// TIA Portal V17 export
// export: Created 2025-06-26T07:49:37.0369601Z, ExportSetting WithDefaults, DisplayName Totally Integrated Automation Portal, DisplayVersion V17 Update 8, DisplayName TIA Portal Openness, DisplayVersion V17 Update 8, DisplayName TIA Portal Version Control Interface, DisplayVersion V17, DisplayName STEP 7 Professional, DisplayVersion V17 Update 8, DisplayName STEP 7 Safety, DisplayVersion V17 Update 6, DisplayName WinCC Advanced, DisplayVersion V17 Update 8
FUNCTION "Control" : Void   // FC3, FBD
TITLE = Sequencing of control algorithms
{ S7_Optimized_Access := 'TRUE' }
AUTHOR : Heaten
VERSION : 0.1
// stored: AutoNumber true, IsIECCheckEnabled false, SetENOAutomatically false, UDAEnableTagReadback false
BEGIN

REGION Network 1: Calculations for process controlling and monitoring
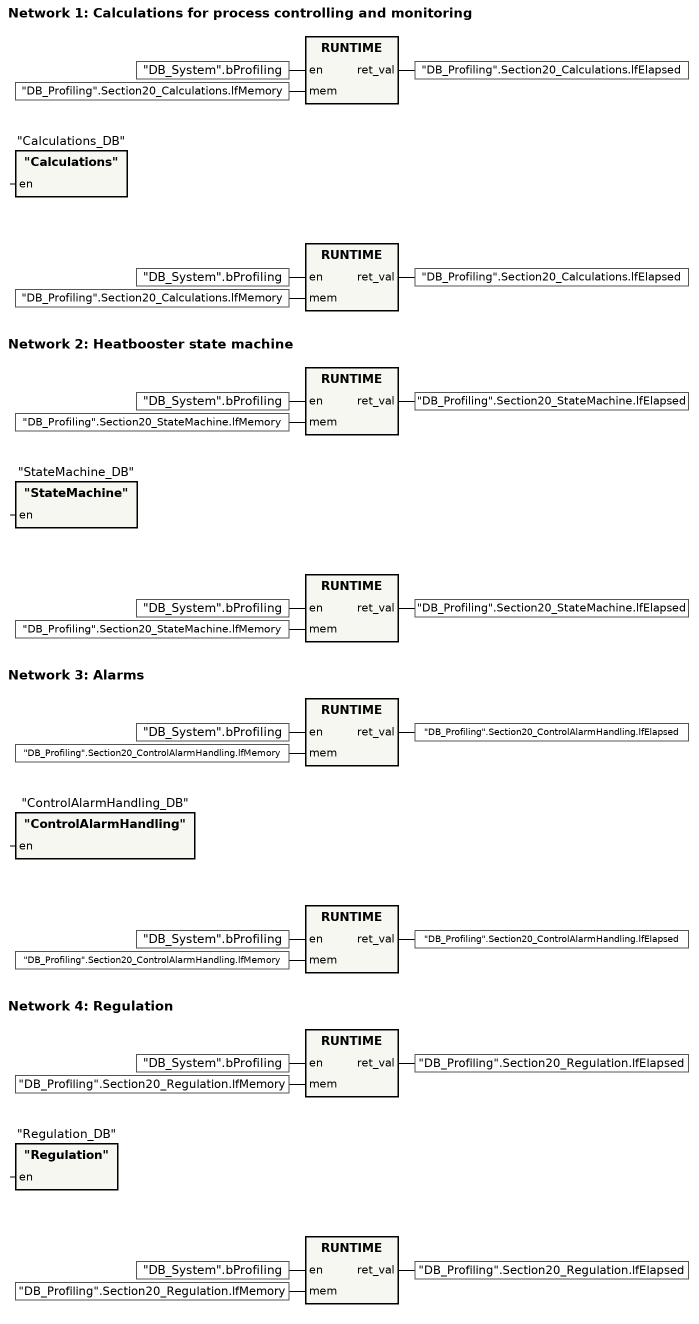
   // no SCL statement known for Runtime: written as a call
   IF "DB_System".bProfiling THEN
       "DB_Profiling".Section20_Calculations.lfElapsed := Runtime(mem := "DB_Profiling".Section20_Calculations.lfMemory);
   END_IF;
   "Calculations_DB"();   // "Calculations"
   IF "DB_System".bProfiling THEN
       "DB_Profiling".Section20_Calculations.lfElapsed := Runtime(mem := "DB_Profiling".Section20_Calculations.lfMemory);
   END_IF;
END_REGION

REGION Network 2: Heatbooster state machine
   // no SCL statement known for Runtime: written as a call
   IF "DB_System".bProfiling THEN
       "DB_Profiling".Section20_StateMachine.lfElapsed := Runtime(mem := "DB_Profiling".Section20_StateMachine.lfMemory);
   END_IF;
   "StateMachine_DB"();   // "StateMachine"
   IF "DB_System".bProfiling THEN
       "DB_Profiling".Section20_StateMachine.lfElapsed := Runtime(mem := "DB_Profiling".Section20_StateMachine.lfMemory);
   END_IF;
END_REGION

REGION Network 3: Alarms
   // no SCL statement known for Runtime: written as a call
   IF "DB_System".bProfiling THEN
       "DB_Profiling".Section20_ControlAlarmHandling.lfElapsed := Runtime(mem := "DB_Profiling".Section20_ControlAlarmHandling.lfMemory);
   END_IF;
   "ControlAlarmHandling_DB"();   // "ControlAlarmHandling"
   IF "DB_System".bProfiling THEN
       "DB_Profiling".Section20_ControlAlarmHandling.lfElapsed := Runtime(mem := "DB_Profiling".Section20_ControlAlarmHandling.lfMemory);
   END_IF;
END_REGION

REGION Network 4: Regulation
   // no SCL statement known for Runtime: written as a call
   IF "DB_System".bProfiling THEN
       "DB_Profiling".Section20_Regulation.lfElapsed := Runtime(mem := "DB_Profiling".Section20_Regulation.lfMemory);
   END_IF;
   "Regulation_DB"();   // "Regulation"
   IF "DB_System".bProfiling THEN
       "DB_Profiling".Section20_Regulation.lfElapsed := Runtime(mem := "DB_Profiling".Section20_Regulation.lfMemory);
   END_IF;
END_REGION

REGION Network 5: Start and stop
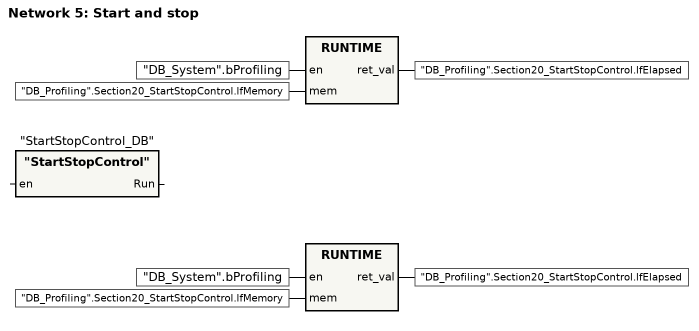
   // no SCL statement known for Runtime: written as a call
   IF "DB_System".bProfiling THEN
       "DB_Profiling".Section20_StartStopControl.lfElapsed := Runtime(mem := "DB_Profiling".Section20_StartStopControl.lfMemory);
   END_IF;
   "StartStopControl_DB"();   // "StartStopControl"
   IF "DB_System".bProfiling THEN
       "DB_Profiling".Section20_StartStopControl.lfElapsed := Runtime(mem := "DB_Profiling".Section20_StartStopControl.lfMemory);
   END_IF;
END_REGION
END_FUNCTION
